PROGRAM MAIN
VAR
	fbHttp_ClientPost	: FB_Http_Client;
	stHttpReqPost		: ST_HTTP_Request; 
	stHttpResponsePost	: ST_HTTP_Response;
	sResponsePost		: STRING(255);
	T1_TON				: TON;
	
	fbHttp_ClientGet	: FB_Http_Client;
	stHttpReqGet		: ST_HTTP_Request; 
	stHttpResponseGet	: ST_HTTP_Response;
	T2_TON				: TON;
	sResponseGet		: STRING(255);
	udCounter			: UDINT;
END_VAR

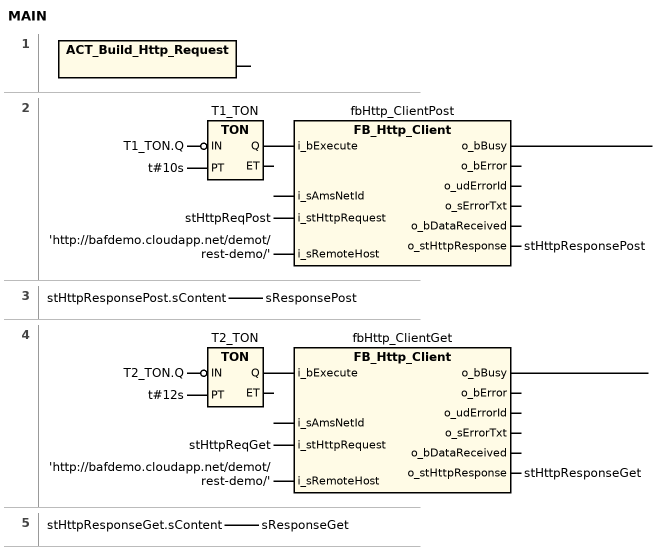
// NETWORK 1
ACT_Build_Http_Request();

// NETWORK 2
T1_TON(IN := NOT T1_TON.Q, PT := t#10s); // TON
fbHttp_ClientPost(
    i_bExecute := T1_TON.Q,
    i_stHttpRequest := stHttpReqPost,
    i_sRemoteHost := 'http://bafdemo.cloudapp.net/demot/rest-demo/',
    o_stHttpResponse => stHttpResponsePost); // FB_Http_Client

// NETWORK 3
sResponsePost := stHttpResponsePost.sContent;

// NETWORK 4
T2_TON(IN := NOT T2_TON.Q, PT := t#12s); // TON
fbHttp_ClientGet(
    i_bExecute := T2_TON.Q,
    i_stHttpRequest := stHttpReqGet,
    i_sRemoteHost := 'http://bafdemo.cloudapp.net/demot/rest-demo/',
    o_stHttpResponse => stHttpResponseGet); // FB_Http_Client

// NETWORK 5
sResponseGet := stHttpResponseGet.sContent;

ACTION ACT_Build_Http_Request:

(****  HTTP POST Example ********************************************************************************)

stHttpReqPost.eHttpRequestType 			:= E_HTTP_Request_Type.E_HTTP_Request_Type_POST;

stHttpReqPost.arrParameters[0].sName	:= 'passwd';
stHttpReqPost.arrParameters[0].sValue	:= 'TwoCats';

stHttpReqPost.arrParameters[1].sName	:= 'counter';
stHttpReqPost.arrParameters[1].sValue	:= UDINT_TO_STRING(udCounter);  udCounter := udCounter + 1;

stHttpReqPost.arrParameters[2].sName	:= 'cyclecount';
stHttpReqPost.arrParameters[2].sValue	:= UDINT_TO_STRING(_TaskInfo[1].CycleCount);

(*******************************************************************************************************)

(****  HTTP GET Example ********************************************************************************)

stHttpReqGet.eHttpRequestType 			:= E_HTTP_Request_Type.E_HTTP_Request_Type_GET;

stHttpReqGet.arrParameters[0].sName		:= 'passwd';
stHttpReqGet.arrParameters[0].sValue	:= 'TwoCats';

stHttpReqGet.arrParameters[1].sName		:= 'parameters';
stHttpReqGet.arrParameters[1].sValue	:= '1';

(*******************************************************************************************************)
END_ACTION

END_PROGRAM

(* stored: Version 1.1.0.1, ProductVersion 3.1.4020.12
   POU MAIN: Id {7157c66d-973e-4a2d-8457-3b82a89435c7}, SpecialFunc None
   Action ACT_Build_Http_Request: Id {cc5077de-76fe-4954-9bf1-47dba06f345a} *)
